PROGRAM stopping_mode
VAR
	ed_routine_stopping_idle: BOOL;
	stack_power_enabled: BOOL;
	RECTIFIER_OUTPUT_OFF: BOOL;// ADD LOGIC FOR MONITORING RECTIFIER OUTPUT - USE CT? VERIFY PS DOES NOT MOVE CURRENT WHEN POWERED OFF
	u_3112_stop_request: BOOL;
	u_3212_stop_request: BOOL;
	u_3312_stop_request: BOOL;
	u_3405_stop_request: BOOL;
	u_3160_stop_request: BOOL
;
	u_3260_stop_request: BOOL;
	u_3360_stop_request: BOOL;
	u_3370_stop_request: BOOL;
	u_3112_run_feedback: BOOL;
	u_3212_run_feedback: BOOL;
	u_3312_run_feedback: BOOL;
	u_3405_run_feedback: BOOL;
	u_3160_run_feedback: BOOL;
	u_3260_run_feedback: BOOL;
	u_3360_run_feedback: BOOL;
	u_3370_run_feedback: BOOL;
	
	nv_3110_stop_request:BOOL;
	av_3248_stop_request: BOOL;
	av_3148_stop_request: BOOL;
	nv_3335_stop_request: BOOL;
	nv_3235_stop_request: BOOL;
	nv_3135_stop_request: BOOL;
	nv_3310_stop_request: BOOL;
	nv_3210_stop_request: BOOL;
	ed_routine_stop_mode: BOOL;
	redox_doser_stop_request: BOOL;
	nv_3335_position_request: INT;
	av_3148_position_request: INT;
	av_3248_position_request: INT;
	ed_pumps_stopped: BOOL;
	nv_3110_closed_feedback: BOOL;
	nv_3210_closed_feedback: BOOL;
	nv_3310_closed_feedback: BOOL;
	nv_3135_closed_feedback: BOOL;
	nv_3235_closed_feedback: BOOL;
	nv_3335_position_feedback: INT;
	nv_3335_recycle_position: BOOL;
	av_3148_position_feedback: INT;
	av_3148_recycle_position: BOOL;
	av_3248_recycle_position: BOOL;
	ed_valves_stopped: BOOL;
	ed_stopped: BOOL;
	av_3348_position_request: INT;
	nv_3372_stop_request: BOOL;
	av_3348_position_feedback: INT;
	av_3348_recycle_position: BOOL;
	nv_3335_closed_feedback: BOOL;
	nv_3372_closed_feedback: BOOL;
	nv_3162_stop_request: BOOL;
	ed_critical_stop: BOOL;
	tmr_stop_pump_delay: TON;
	tmr_stop_pump_delay_pt: TIME := T#10S;
	tmr_stop_pump_delay_et: TIME;
END_VAR
VAR // added by the converter: edge detectors and wires of the graphical bodies
    _w1, _w2, _w3 : BOOL;
END_VAR

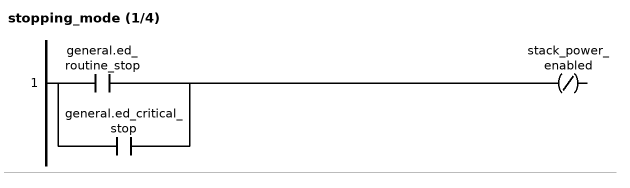
// NETWORK 1
stack_power_enabled := NOT (general.ed_routine_stop OR general.ed_critical_stop);

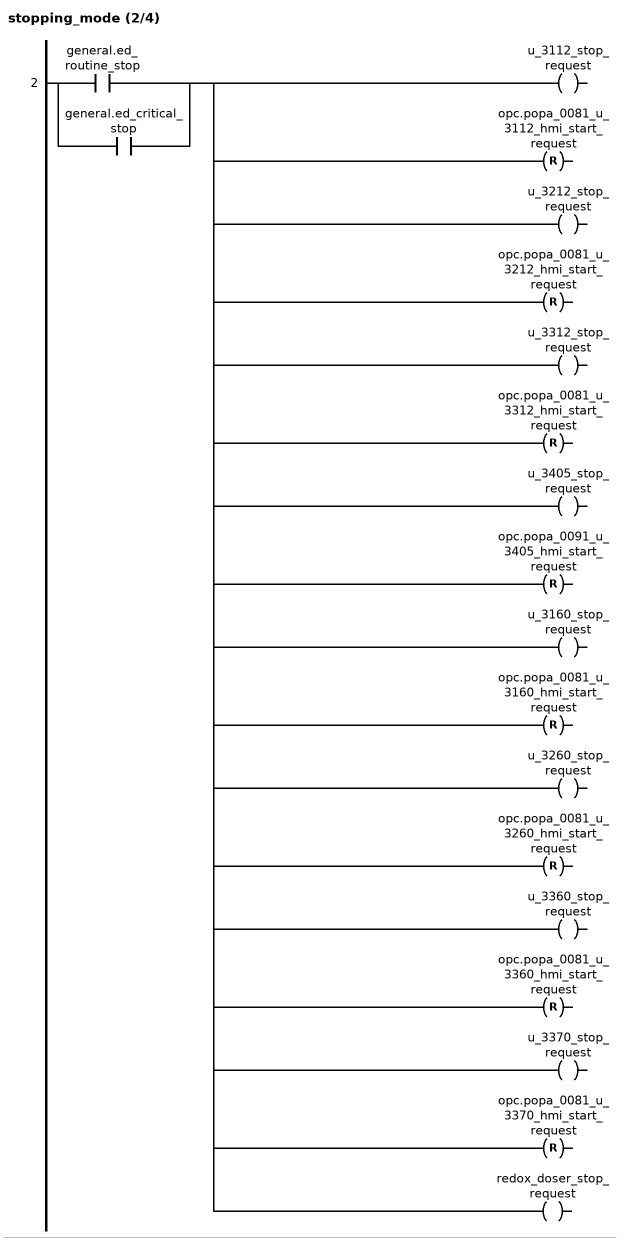
// NETWORK 2
_w1 := general.ed_routine_stop OR general.ed_critical_stop;
u_3112_stop_request := _w1;
opc.popa_0081_u_3112_hmi_start_request R= _w1;
u_3212_stop_request := _w1;
opc.popa_0081_u_3212_hmi_start_request R= _w1;
u_3312_stop_request := _w1;
opc.popa_0081_u_3312_hmi_start_request R= _w1;
u_3405_stop_request := _w1;
opc.popa_0091_u_3405_hmi_start_request R= _w1;
u_3160_stop_request := _w1;
opc.popa_0081_u_3160_hmi_start_request R= _w1;
u_3260_stop_request := _w1;
opc.popa_0081_u_3260_hmi_start_request R= _w1;
u_3360_stop_request := _w1;
opc.popa_0081_u_3360_hmi_start_request R= _w1;
u_3370_stop_request := _w1;
opc.popa_0081_u_3370_hmi_start_request R= _w1;
redox_doser_stop_request := _w1;

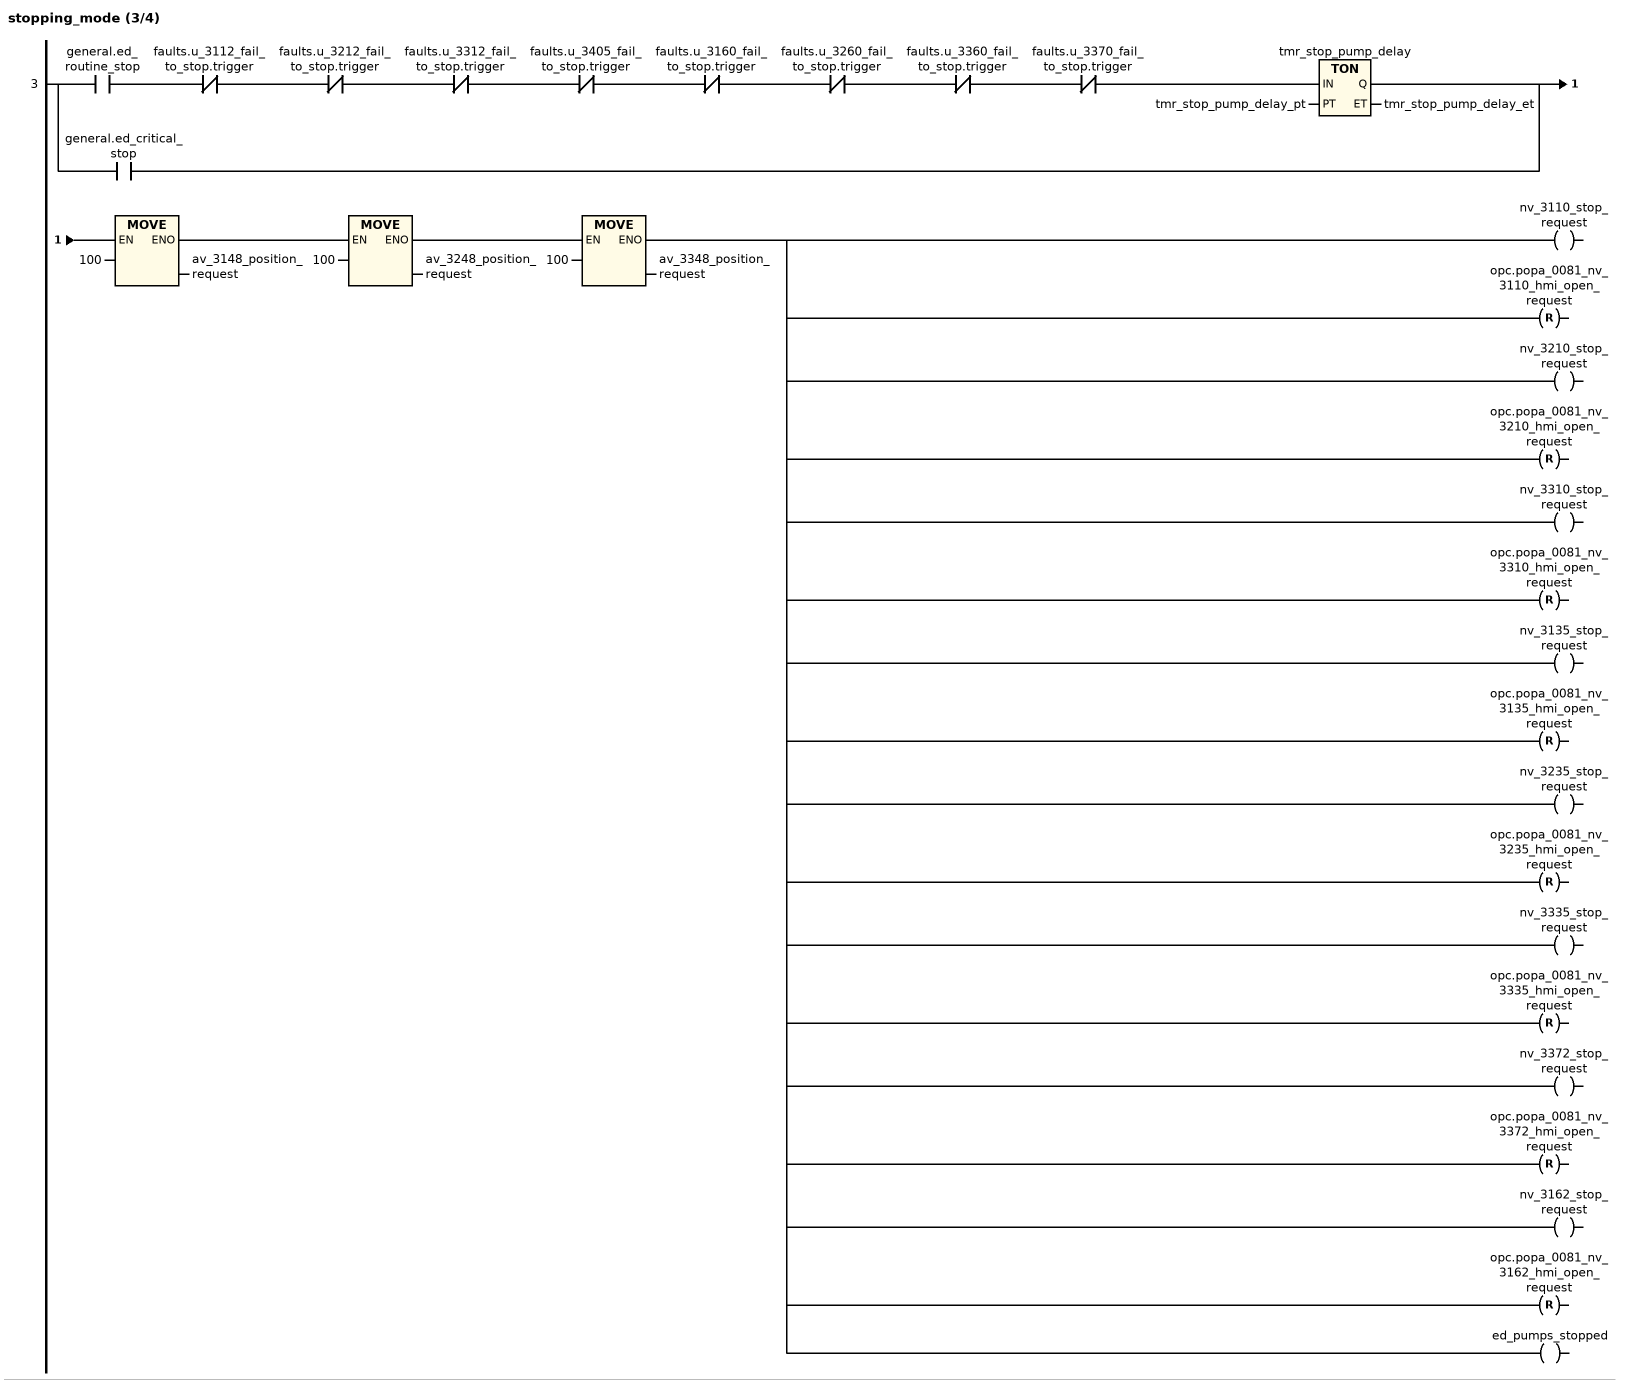
// NETWORK 3
tmr_stop_pump_delay(
    IN := general.ed_routine_stop AND NOT faults.u_3112_fail_to_stop.trigger AND NOT faults.u_3212_fail_to_stop.trigger AND NOT faults.u_3312_fail_to_stop.trigger AND NOT faults.u_3405_fail_to_stop.trigger AND NOT faults.u_3160_fail_to_stop.trigger AND NOT faults.u_3260_fail_to_stop.trigger AND NOT faults.u_3360_fail_to_stop.trigger AND NOT faults.u_3370_fail_to_stop.trigger,
    PT := tmr_stop_pump_delay_pt,
    ET => tmr_stop_pump_delay_et); // TON
_w2 := tmr_stop_pump_delay.Q OR general.ed_critical_stop;
IF _w2 THEN av_3148_position_request := 100; END_IF
IF _w2 THEN av_3248_position_request := 100; END_IF
IF _w2 THEN av_3348_position_request := 100; END_IF
nv_3110_stop_request := _w2;
opc.popa_0081_nv_3110_hmi_open_request R= _w2;
nv_3210_stop_request := _w2;
opc.popa_0081_nv_3210_hmi_open_request R= _w2;
nv_3310_stop_request := _w2;
opc.popa_0081_nv_3310_hmi_open_request R= _w2;
nv_3135_stop_request := _w2;
opc.popa_0081_nv_3135_hmi_open_request R= _w2;
nv_3235_stop_request := _w2;
opc.popa_0081_nv_3235_hmi_open_request R= _w2;
nv_3335_stop_request := _w2;
opc.popa_0081_nv_3335_hmi_open_request R= _w2;
nv_3372_stop_request := _w2;
opc.popa_0081_nv_3372_hmi_open_request R= _w2;
nv_3162_stop_request := _w2;
opc.popa_0081_nv_3162_hmi_open_request R= _w2;
ed_pumps_stopped := _w2;

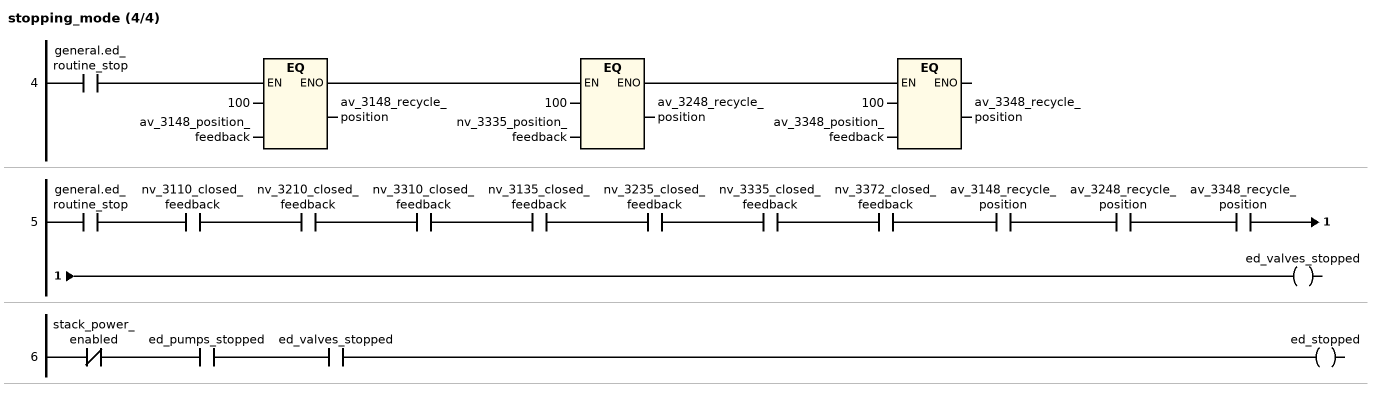
// NETWORK 4
_w3 := general.ed_routine_stop;
IF _w3 THEN av_3148_recycle_position := 100 = av_3148_position_feedback; END_IF
IF _w3 THEN av_3248_recycle_position := 100 = nv_3335_position_feedback; END_IF
IF _w3 THEN av_3348_recycle_position := 100 = av_3348_position_feedback; END_IF

// NETWORK 5
ed_valves_stopped := general.ed_routine_stop AND nv_3110_closed_feedback AND nv_3210_closed_feedback AND nv_3310_closed_feedback AND nv_3135_closed_feedback AND nv_3235_closed_feedback AND nv_3335_closed_feedback AND nv_3372_closed_feedback AND av_3148_recycle_position AND av_3248_recycle_position AND av_3348_recycle_position;

// NETWORK 6
ed_stopped := NOT stack_power_enabled AND ed_pumps_stopped AND ed_valves_stopped;

END_PROGRAM

(* stored: Version 1.1.0.1, ProductVersion 3.1.4024.12
   POU stopping_mode: Id {65ab387d-14b6-4597-8712-6f6f31d5a03f}, SpecialFunc None *)
